{attribute 'GeneratedUsingTerminal: EL5042-0000-0016'}
{attribute addProperty BoxType "EL5042-0000-0016"}
{attribute addProperty Id "FB_Inputs_Channel_1AT %I*FB_Inputs_Channel_7405098814FB_Inputs_Channel_2AT %I*FB_Inputs_Channel_7405098814WcStateAT %I*WcState_9091E0EB2InfoDataAT %I*InfoData_32EB74EA10"}
{attribute addProperty CRC "1814315440"}
{attribute addProperty Size "40"}
TYPE EL5042_6C2441B0 :
STRUCT
	{attribute addProperty Name "FB_Inputs_Channel_1"}
	FB_Inputs_Channel_1 : FB_Inputs_Channel_74050988;
	{attribute addProperty Name "FB_Inputs_Channel_2"}
	FB_Inputs_Channel_2 : FB_Inputs_Channel_74050988;
	{attribute addProperty Name "WcState"}
	WcState : WcState_9091E0EB;
	{attribute addProperty Name "InfoData"}
	InfoData : InfoData_32EB74EA;
END_STRUCT
END_TYPE

(* stored: Version 1.2.0.0, ProductVersion 3.1.4024.9
   DUT EL5042_6C2441B0: Id {7ab12004-8097-4155-8730-f034b8529266} *)
